PROGRAM MAIN
VAR
	MachineControll : MachineControlMode ; 
	
END_VAR

MachineControll();

END_PROGRAM

(* stored: Version 1.1.0.1, ProductVersion 3.1.4024.12
   POU MAIN: Id {296c9099-8b07-4824-9c8d-85d794132ef3}, SpecialFunc None *)
